PROGRAM Combined_Vertical
VAR
//Outputs: Power for Limit switches, Home Sensors, etc.
    //bPowerSwitchesAxis1 AT %Q*: BOOL:= TRUE;

//Hardware interlocks
    //bInterlockFwdOK AT %I*: BOOL;
END_VAR

//Initial parameters of an Axis
(*IF _TaskInfo[fbGetCurTaskIndex.index].FirstCycle THEN
    //Initial default values:
    GVL.astAxes[1].stConfig.eHomeSeq := 0;
    GVL.astAxes[1].stConfig.fHomePosition := 0.0;
    GVL.astAxes[1].stConfig.fHomeFinishDistance := 0.0;
    GVL.astAxes[1].stConfig.eRestorePosition := E_RestorePosition.eRestoreWithoutHome;
END_IF*)

//Define ACTIONS() or write exclusive code for an specific axis.
(*Eg. Stop when temperature reaches certain values, reduce speed if  a signal is activated, etc.
Eg. GVL.astAxes[x].stControl.bInterlockFwd := NOT bInterlockFwdOK;*)


(*
This will be the axis that drives the vertical stages, there will be no "real master"
This axis will only be able to run if the two axes below it are coupled in.
*)

END_PROGRAM

(* stored: Version 1.1.0.1, ProductVersion 3.1.4024.11
   POU Combined_Vertical: Id {0f34f732-07ed-43ff-ba09-f9229513977f}, SpecialFunc None *)
